{attribute addProperty BoxType "EP6224-0002-0016"}
{attribute addProperty Id "DI_X01_Pin2AT %I*BOOL811DI_X02_Pin2AT %I*BOOL812DI_X03_Pin2AT %I*BOOL813DI_X04_Pin2AT %I*BOOL814"}
{attribute addProperty CRC "1030352877"}
{attribute addProperty SizeInBites "32"}
{attribute addProperty SizeInBytes "4"}
TYPE Digital_Inputs_3D69EFED :
STRUCT
	{attribute addProperty Name "DI_X01_Pin2"}
	DI_X01_Pin2 AT %I* : BOOL;
	{attribute addProperty Name "DI_X02_Pin2"}
	DI_X02_Pin2 AT %I* : BOOL;
	{attribute addProperty Name "DI_X03_Pin2"}
	DI_X03_Pin2 AT %I* : BOOL;
	{attribute addProperty Name "DI_X04_Pin2"}
	DI_X04_Pin2 AT %I* : BOOL;
END_STRUCT
END_TYPE

(* stored: Version 1.2.0.0, ProductVersion 3.1.4024.9
   DUT Digital_Inputs_3D69EFED: Id {b976357a-de06-4e97-a904-0a0492c8cb4e} *)
